		IF GVL_MOTION.STOP_INT THEN
			GVL_MOTION.STATUS.Stop_Int							:= TRUE;
			GVL_MOTION.xCon.Execute_MABS 						:= FALSE;
			GVL_MOTION.yCon.Execute_MABS 						:= FALSE;
			GVL_MOTION.zCon.Execute_MABS 						:= FALSE;
			GVL_MOTION.xCon.Execute_MREL 						:= FALSE;
			GVL_MOTION.yCon.Execute_MREL 						:= FALSE;	
			GVL_MOTION.zCon.Execute_MREL 						:= FALSE;
			GVL_MOTION.xCon.Execute_HALT 						:= TRUE;
			GVL_MOTION.yCon.Execute_HALT 						:= TRUE;
			GVL_MOTION.zCon.Execute_HALT 						:= TRUE;			
				
			GVL_MOTION.InstructionState 						:= 2;
			t5(IN := FALSE);
			
		
		//with no timer pause in between instructions MoveDone stays high long enough to skip an instruction
		//instruction always loaded but queue index is skipped
		ELSIF GVL_MOTION.xOut.MoveDone AND GVL_MOTION.yOut.MoveDone AND GVL_MOTION.zOut.MoveDone THEN //these signals depend on execute MABS/MREL
		
			timer(IN := TRUE, PT := T#1MS);
			
			IF timer.Q THEN
				GVL_MOTION.xCon.Execute_MABS 					:= FALSE;
				GVL_MOTION.xCon.Execute_MREL 					:= FALSE;
				GVL_MOTION.yCon.Execute_MABS 					:= FALSE;
				GVL_MOTION.yCon.Execute_MREL 					:= FALSE;	
				GVL_MOTION.zCon.Execute_MABS 					:= FALSE;
				GVL_MOTION.zCon.Execute_MREL 					:= FALSE;		
				timer(IN := FALSE);
				
				IF GVL_MOTION.CurInstruction < (GVL_MOTION.ScriptEnd - 1) THEN
					GVL_MOTION.CurInstruction 					:= GVL_MOTION.CurInstruction + 1; //queue next instruction
					GVL_MOTION.InstructionState 				:= 0;
					t5(IN := FALSE);
				ELSE
					GVL_MOTION.CurInstruction 					:= 0;
					GVL_MOTION.InstructionState 				:= 0;
					t5(IN := FALSE);
					IF NOT GVL_MOTION.EXT_CTR.CMDLOOP THEN
						IF GVL_MOTION.RUN_INDEX >= GVL_MOTION.EXT_CTR.SCRIPTITERATIONS THEN
							GVL_MOTION.RUN_INDEX				:= 1;
							GVL_MOTION.EXT_CTR.CMDRUN 			:= FALSE;	 //command list executed
						ELSE
							GVL_MOTION.RUN_INDEX				:= GVL_MOTION.RUN_INDEX + 1;	
						END_IF
						
					ELSE
						
						GVL_MOTION.RUN_INDEX					:= GVL_MOTION.RUN_INDEX + 1;
					END_IF
					
				END_IF
				
			END_IF	
			
		END_IF
	
	END_IF
	
	2:
	//state 2: pause motion
	//debounce timer
	t4(IN := TRUE, PT := T#30MS);
	
	
	IF t4.Q THEN
		IF GVL_MOTION.STOP_INT THEN
			GVL_MOTION.STATUS.Stop_Int							:= FALSE; //lamp off
			GVL_MOTION.xCon.Execute_HALT 						:= FALSE;
			GVL_MOTION.yCon.Execute_HALT 						:= FALSE;
			GVL_MOTION.zCon.Execute_HALT 						:= FALSE;
			
			IF GVL_MOTION.Script[GVL_MOTION.CurInstruction].MotionCommand = MotionType.Absolute THEN	
				GVL_MOTION.xCon.Execute_MABS 					:= TRUE;
				GVL_MOTION.yCon.Execute_MABS 					:= TRUE;		
				GVL_MOTION.zCon.Execute_MABS 					:= TRUE;
			
				GVL_MOTION.InstructionState 					:= 1;	
				t4(IN := FALSE);
				
			ELSIF GVL_MOTION.Script[GVL_MOTION.CurInstruction].MotionCommand = MotionType.Relative THEN
				GVL_MOTION.xCon.Execute_MREL 					:= TRUE;
				GVL_MOTION.yCon.Execute_MREL 					:= TRUE;
				GVL_MOTION.zCon.Execute_MREL 					:= TRUE;
			
				GVL_MOTION.InstructionState 			  		:= 1;	
				t4(IN := FALSE);
				
			ELSIF GVL_MOTION.Script[GVL_MOTION.CurInstruction].MotionCommand = MotionType.Time_Wait THEN	
				t2(IN := TRUE, PT := hold);
				GVL_MOTION.InstructionState						:= 3;
			ELSE
				error											:= TRUE;
			END_IF
		
		END_IF
	
	END_IF
	
	3:
	//state 3: timed pause. 
	IF GVL_MOTION.STOP_INT THEN
		GVL_MOTION.STATUS.Stop_Int								:= TRUE; //lamp on
		hold													:= GVL_MOTION.Script[GVL_MOTION.CurInstruction].PauseTime - t2.ET;
		t2(IN := FALSE);
		GVL_MOTION.InstructionState								:= 2;
	ELSIF t2.Q THEN
		t2(IN := FALSE);
		IF GVL_MOTION.CurInstruction < (GVL_MOTION.ScriptEnd - 1) THEN
			GVL_MOTION.CurInstruction 							:= GVL_MOTION.CurInstruction + 1; //queue next instruction
			GVL_MOTION.InstructionState 						:= 0;
					
		ELSE
			GVL_MOTION.CurInstruction 							:= 0;
			GVL_MOTION.InstructionState 						:= 0;
			t5(IN := FALSE);
			IF NOT GVL_MOTION.EXT_CTR.CMDLOOP THEN
				IF GVL_MOTION.RUN_INDEX >= GVL_MOTION.EXT_CTR.SCRIPTITERATIONS THEN
					GVL_MOTION.RUN_INDEX						:= 1;
					GVL_MOTION.EXT_CTR.CMDRUN 					:= FALSE;	 //command list executed
				ELSE
					GVL_MOTION.RUN_INDEX						:= GVL_MOTION.RUN_INDEX + 1;	
				END_IF
				
			ELSE
			
				GVL_MOTION.RUN_INDEX							:= GVL_MOTION.RUN_INDEX + 1;
			END_IF
			
		END_IF
	ELSE
		error													:= TRUE;	
	END_IF
		
END_CASE

END_PROGRAM

// ---- POUs/HomeFixRack.TcPOU
PROGRAM HomeFixRack
VAR
END_VAR

CASE GVL_MOTION.HomingState OF
	0:
	GVL_MOTION.zCon.Execute_HOME			:= TRUE;
	GVL_MOTION.HomingState					:= 1;
	
	1:
	IF GVL_MOTION.zHomeStatus.Done THEN
		GVL_MOTION.zCon.Execute_HOME		:= FALSE;
		GVL_MOTION.yCon.Execute_HOME		:= TRUE;
		GVL_MOTION.HomingState				:= 2;
	END_IF
	
	2:
	IF GVL_MOTION.yHomeStatus.Done THEN
		GVL_MOTION.yCon.Execute_HOME		:= FALSE;
		IF NOT GVL_MOTION.xOut.AxisCoupled THEN
			GVL_MOTION.xCon.ExecuteUncouple	:= FALSE;
			GVL_MOTION.xCon.ExecuteCouple	:= TRUE;
		END_IF
		
		GVL_MOTION.HomingState				:= 3;
	END_IF
	
	3:
	IF GVL_MOTION.xOut.AxisCoupled THEN
		GVL_MOTION.xJogBW					:= TRUE;
		GVL_MOTION.HomingState				:= 4;
	END_IF
	
	4:
	IF GVL_MOTION.xCon.LimNeg OR GVL_MOTION.xcCon.LimNeg THEN
		GVL_MOTION.xJogBW					:= FALSE;
		GVL_MOTION.xCon.SetPosition			:= 5;
		GVL_MOTION.xCon.SetVelocity			:= 50;
		
		GVL_MOTION.HomingState				:= 5;
	
	END_IF
	
	5:
	GVL_MOTION.xCon.Execute_MREL			:= TRUE;
	GVL_MOTION.HomingState					:= 6;	
	
	6:
	IF GVL_MOTION.xOut.MoveDone THEN
		GVL_MOTION.xCon.Execute_MREL		:= FALSE;
		GVL_MOTION.xCon.ExecuteCouple		:= FALSE;
		GVL_MOTION.xCon.ExecuteUncouple 	:= TRUE;
		GVL_MOTION.HomingState				:= 7;
	END_IF
	
	7:
	IF NOT GVL_MOTION.xOut.AxisCoupled THEN
		GVL_MOTION.xCon.Execute_HOME		:= TRUE; 
		GVL_MOTION.HomingState				:= 8;
	END_IF
	
	8:
	IF GVL_MOTION.xHomeStatus.Done THEN
		GVL_MOTION.xCon.Execute_HOME		:= FALSE;
		GVL_MOTION.xcCon.Execute_HOME		:= TRUE;
 		GVL_MOTION.HomingState				:= 9;
	END_IF
	
	9:
	IF GVL_MOTION.xcHomeStatus.Done THEN
		GVL_MOTION.xcCon.Execute_HOME		:= FALSE;
		GVL_MOTION.xCon.ExecuteUncouple 	:= FALSE;
		GVL_MOTION.HomingState				:= 10;
	END_IF
	
	10:
	GVL_MOTION.HomingState					:= 0;
	GVL_MOTION.xCon.ExecuteCouple			:= TRUE;
	GVL_MOTION.AxesLocated					:= TRUE;
	GVL_MOTION.EXT_CTR.CMDHOME				:= FALSE;
END_CASE

END_PROGRAM

// ---- POUs/RackCheck.TcPOU
PROGRAM RackCheck
VAR
	state		:INT	:= 0;
	tempX1		:LREAL;
	tempX2		:LREAL;
	compare		:LREAL;
END_VAR

CASE state OF
	0: //direction of motion unknown
		IF GVL_MOTION.NPNX THEN
			tempX1								:= GVL_MOTION.xOut.PositionOut;
			state								:= 1;
		ELSIF GVL_MOTION.NPNXC THEN	
			tempX1								:= GVL_MOTION.xOut.PositionOut;
			state								:= 2;
		END_IF
		
	1:
		IF GVL_MOTION.NPNXC THEN
			tempX2	:= GVL_MOTION.xOut.PositionOut;
			compare	:= tempX1 - tempX2;
			IF compare > 5 THEN //XC ahead, negative motion
				GVL_MOTION.STATUS.Rack_Err		:= TRUE;
				state							:= 3;
			ELSIF compare < -5 THEN //X ahead, positive motion
				GVL_MOTION.STATUS.Rack_Err		:= TRUE;
				state							:= 3;
			ELSE
				state							:= 0;	
			END_IF
		END_IF	
		
	2:
		IF GVL_MOTION.NPNX THEN
			tempX2								:= GVL_MOTION.xOut.PositionOut;
			compare								:= tempX2 - tempX1;
			IF compare > 5 THEN //XC ahead, positive motion
				GVL_MOTION.STATUS.Rack_Err		:= TRUE;
				state							:= 3;
			ELSIF compare < -5 THEN //X ahead, negative motion
				GVL_MOTION.STATUS.Rack_Err		:= TRUE;
				state							:= 3;
			ELSE
				state							:= 0;	
			END_IF
		END_IF
		
	3: //move X relative by compare
		IF GVL_MOTION.EXT_CTR.CMDFIXRACK AND NOT GVL_MOTION.EXT_CTR.CMDRUN THEN
			GVL_MOTION.xCon.SetPosition			:= compare;
			GVL_MOTION.xCon.ExecuteUncouple		:= TRUE;
			IF NOT GVL_MOTION.xOut.AxisCoupled THEN
				GVL_MOTION.EXT_CTR.CMDFIXRACK	:= FALSE;
				GVL_MOTION.xCon.Execute_MREL	:= TRUE;
				state							:= 4;
			END_IF
		END_IF
	
	4:
		IF GVL_MOTION.xOut.MoveDone THEN
			GVL_MOTION.xCon.Execute_MREL	:= FALSE;
			GVL_MOTION.STATUS.Rack_Err		:= FALSE;
			state							:= 0;
		END_IF
END_CASE

END_PROGRAM

// ---- GlobalTextList.TcGTLO
TEXTLIST GlobalTextList
  803 = '%.0f'
  981 = '%.4f'
  59 = '%4d'
  1444 = '%5d'
  184 = '%s'
  530 = '%t'
  653 = '& Continue From Fault'
  797 = '(Lower Limit)'
  639 = '5'
  56 = '50'
  371 = '500'
  280 = '<- NOT IMPLEMENTED'
  2 = 'A'
  231 = 'ABSOLUTE POSITION'
  461 = 'ACCEL/DECEL'
  34 = 'Accel/Decel'
  466 = 'ACCELERATING'
  532 = 'Actual Position'
  447 = 'Actual Speed'
  575 = 'Add Command to Queue'
  1059 = 'Add Instruction to Script'
  263 = 'AddCMDtoQueue'
  847 = 'AddCMDtoQuue'
  55 = 'Administrator'
  1058 = 'Append Data (single CSV)'
  1775 = 'Axes Located'
  640 = 'Axis to Trigger On'
  687 = 'Axis to Trigger On (NO SICK)'
  2271 = 'B'
  1705 = 'Basin Control'
  458 = 'Basin CTR'
  1413 = 'Basin Set'
  100 = 'BROKEN'
  1205 = 'Capture Data Every X MM'
  869 = 'Capture Data Every X MM/S'
  1220 = 'Clear Data'
  273 = 'Clear Loaded Script'
  848 = 'Clear Queue'
  888 = 'CLICK TO CONTINUE'
  1102 = 'CMD'
  58 = 'CMDtoAdd'
  561 = 'Command'
  312 = 'Command type'
  855 = 'Command Type'
  616 = 'Comment'
  899 = 'Continue From Error'
  293 = 'Continue From Fault'
  313 = 'Continuous Mode'
  1032 = 'Continuous Mode (not for DAQ)'
  101 = 'ContinuousMode'
  425 = 'Couple X Axes'
  416 = 'Current Instruction'
  698 = 'Current Script Run'
  628 = 'DECELERATING'
  1223 = 'Default Basin (Full Area)'
  1420 = 'Delete Last Instruction'
  1786 = 'Delete Loaded Script'
  2013 = 'delete script file'
  140 = 'Delete Script File'
  276 = 'Drive Control'
  485 = 'DRIVE ENABLE'
  614 = 'Drive Error Reset'
  991 = 'E STOP'
  695 = 'ENABLE ALL AXES'
  1622 = 'Enter Comment'
  752 = 'Enter name of basin (no spaces or < > : " / \\ | ? *)'
  1184 = 'Enter Name of Run'
  833 = 'Enter Name of Script'
  326 = 'Enter Name of Script (no spaces or < > : " / \\ | ? *'
  1 = 'Enter Name of Script (no spaces or < > : " / \\ | ? *)'
  1503 = 'Enter Title of Script (no spaces or < > : " / \\ | ? *)'
  958 = 'FAULT RESET'
  745 = 'Fault Reset'
  1527 = 'Fix Rack'
  862 = 'GroupBox'
  665 = 'GVL_MOTION.CommandQueueArray[GVL_MOTION.QueueCur].PauseTime'
  959 = 'Halt'
  241 = 'HaltTime(ms)'
  57 = 'HaltTime(T#XSYMS)'
  95 = 'Home'
  317 = 'Home Both X'
  682 = 'Home Coupled X'
  72 = 'Home Established'
  292 = 'Home X'
  342 = 'Home X (both)'
  733 = 'Home X (not working)'
  1179 = 'Home XYZ'
  846 = 'Home Y'
  185 = 'Home Z'
  689 = 'Homing Routine'
  196 = 'IN POSITION'
  448 = 'IN VELOCITY'
  863 = 'Jog Controls'
  831 = 'k'
  21 = 'Keyence'
  998 = 'Label'
  2027 = 'list'
  420 = 'Locate Hard Stops'
  301 = 'Locate Stops'
  720 = 'Locate Stops NOT IMPLEMENTED'
  712 = 'm'
  245 = 'Main '
  130 = 'Main Sensoor'
  772 = 'Main Sensor'
  605 = 'Main Sensor for DAQ'
  281 = 'Massa'
  319 = 'Motion'
  786 = 'motion cmd'
  1691 = 'Motion CMD'
  545 = 'MOVE ABS EN'
  566 = 'MOVE ACTIVE'
  277 = 'MoveAbsEn'
  632 = 'MOVING'
  1349 = 'Next Instruction'
  633 = 'NOT IMPLEMENTED'
  254 = 'Note: carriage offsets added to these values'
  320 = 'Number of Script Runs'
  1704 = 'Pause'
  457 = 'Pause & WaitOK'
  68 = 'Pause & WaitOK &'
  97 = 'Pause & WaitOK & Continue From Fault'
  105 = 'Pause Motion'
  582 = 'pause time'
  1146 = 'PauseTime'
  818 = 'POSITION'
  473 = 'Position'
  452 = 'Position(AbsorRel'
  926 = 'Position(AbsorRel)'
  996 = 'Position(AbsorRel)(mm)'
  776 = 'PWR Fail'
  787 = 'Rack Error'
  1800 = 'Rackk Error'
  438 = 'Read Script (data/basin/script)'
  634 = 'Read Script (from title)'
  1797 = 'Read Script From File(data/basin/script)'
  419 = 'RELAT'
  676 = 'RELATIVE POSITION'
  572 = 'RESET ALL AXES'
  489 = 'Reset CSV Write'
  162 = 'Reset Enable Error'
  677 = 'REV'
  795 = 'Reverse Couple X'
  719 = 'Run \tQueue'
  999 = 'Run /nQueue'
  256 = 'Run Queue'
  201 = 'RUN QUEUE'
  1126 = 'RUN SCRIPT'
  910 = 'Run Script Continuously'
  785 = 's'
  771 = 'Safe Z Established'
  2090 = 'scriptlist'
  706 = 'Send'
  1909 = 'send list of script names'
  773 = 'send script'
  427 = 'Send To'
  533 = 'Sensor'
  187 = 'Sensors to Record'
  558 = 'Set Basin'
  1079 = 'Set Basin Manually'
  160 = 'Set Safe Z'
  1541 = 'Set Safe Z (lower limit)'
  621 = 'SET SAFE Z FIRST!!'
  1734 = 'Set X'
  53 = 'set x acc'
  1107 = 'set x pos'
  527 = 'set x vel'
  88 = 'Set X Zero'
  717 = 'Set Y'
  1043 = 'set y acc'
  1171 = 'set y pos'
  916 = 'set y vel'
  486 = 'Set Y Zero'
  983 = 'Set Z'
  544 = 'set z pos'
  401 = 'set z vel'
  373 = 'Set Zero'
  604 = 'SICK'
  1746 = 'SICK (X axis)'
  718 = 'SICK (x axis)'
  697 = 'Sonar'
  793 = 'SPEED'
  854 = 'STATIONARY'
  412 = 'STD'
  838 = 'STOP MOTION'
  474 = 'Test for sick (ADS)'
  700 = 'Trigger'
  615 = 'Trigger On'
  1091 = 'Use Basin Coordinates'
  560 = 'Velocity'
  15 = 'VELOCITY CONTROL'
  47 = 'Write Data Test'
  1372 = 'Write Script'
  139 = 'Write Script to File'
  366 = 'X'
  492 = 'x acc'
  129 = 'X Actual Position'
  897 = 'X Actual Speed'
  784 = 'X Coupled Actual Position'
  259 = 'X Coupled Actual Speed'
  901 = 'X Coupled Pos'
  839 = 'X Coupled Spd'
  1675 = 'X Dist to HS'
  2097 = 'X Hard Stop'
  1001 = 'X Max'
  475 = 'X Min'
  511 = 'x pos'
  751 = 'X Position(AbsorRel)(mm)'
  383 = 'x vel'
  885 = 'X Velocity'
  1201 = 'XPos'
  431 = 'xPos'
  255 = 'XVel'
  150 = 'xVel'
  828 = 'xyCMDtoAdd'
  506 = 'xyz motion'
  980 = 'xyzCMDtoAdd'
  1234 = 'xyzMotionCommand'
  906 = 'Y'
  176 = 'y acc'
  746 = 'Y Actual Position'
  547 = 'Y Actual Speed'
  1458 = 'Y Dist to HS'
  1000 = 'Y Hard Stop'
  1376 = 'Y Max'
  215 = 'Y Min'
  982 = 'y pos'
  557 = 'Y Position(AbsorRel)(mm)'
  208 = 'y vel'
  573 = 'Y Velocity'
  559 = 'YPos'
  102 = 'yPos'
  116 = 'YVel'
  8 = 'yVel'
  397 = 'Z'
  509 = 'Z Actual Position'
  504 = 'Z Actual Speed'
  343 = 'z beh'
  432 = 'z brake'
  1751 = 'Z Dist to HS'
  1593 = 'Z Hard Stop'
  631 = 'Z Max'
  1036 = 'Z Min'
  135 = 'z pos'
  972 = 'Z Position(Abs)(mm)'
  662 = 'Z Position(AbsorRel)(mm)'
  125 = 'Z Safe Low'
  1671 = 'z Type'
  636 = 'z vel'
  690 = 'Z Velocity'
  967 = 'zBeh'
  484 = 'zBehavior'
  517 = 'zBehavior (only for xy motion)'
  1119 = 'ZPos'
  49 = 'zPos'
  436 = 'zType'
  1003 = 'ZVel'
  872 = 'zVel'
END_TEXTLIST

// ---- VISUs/visMotorControl.TcVIS
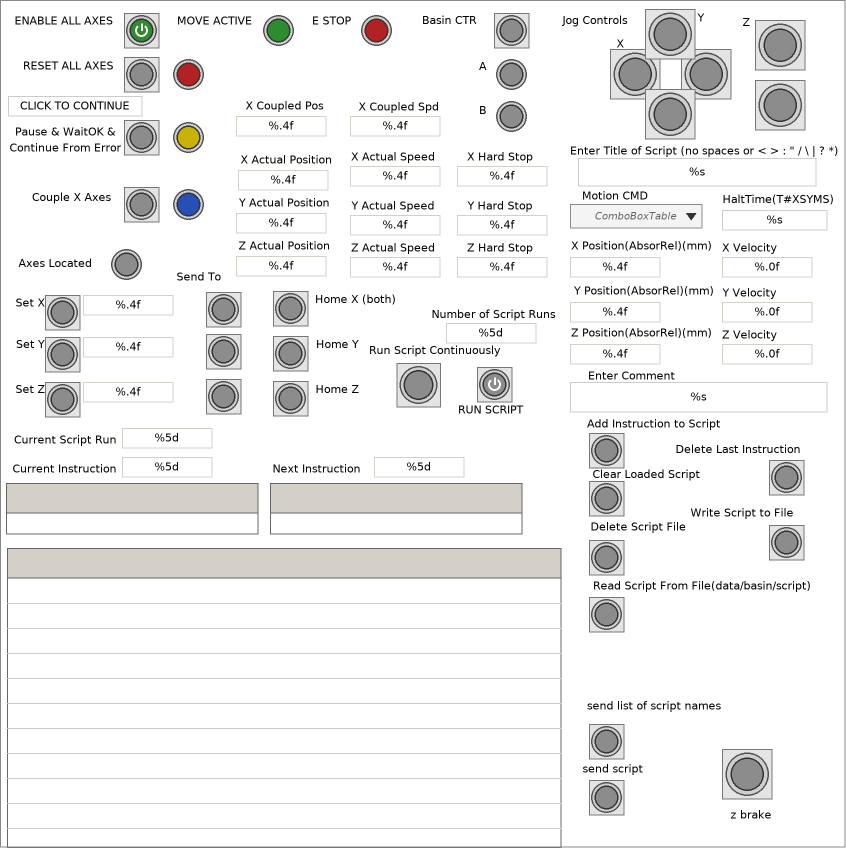
VISUALIZATION visMotorControl  // 846x848
    Label (12,58 113x16), "RESET ALL AXES"
    Label (12,126 107x12), "Pause & WaitOK &"
    Label (9,13 110x16), "ENABLE ALL AXES"
    Textfield (722,257 90x20), "%.0f", text variable: GVL_MOTION.InstructionBuffer.SetXVelocity
        OnMouseClick: write the text variable via InputWithLimits, min 1, max 500, title 'Enter Speed'
    Textfield (570,257 90x20), "%.4f", text variable: GVL_MOTION.InstructionBuffer.SetXPosition
        OnMouseClick: write the text variable via Default, min -200, max 15000
    Label (722,241 55x14), "X Velocity"
    Label (570,238 143x16), "X Position(AbsorRel)(mm)"
    Label (350,149 86x16), "X Actual Speed"
    Label (238,149 97x22), "X Actual Position"
    Textfield (350,166 90x20), "%.4f", text variable: GVL_MOTION.STATUS.xVelOut
    Textfield (238,170 90x20), "%.4f", text variable: GVL_MOTION.STATUS.xPosOut
    ComboBoxTable (570,204 132x24), variable: GVL_MOTION.InstructionBuffer.MotionCommand, data array: GVL_MOTION.xyzCMDSelect
        p1014161805: 4 - 0 + INT#1
        p3854506369: GVL_MOTION.xyzCMDSelect[INDEX]
    Label (564,185 102x22), "Motion CMD"
    PushSwitch (589,433 35x35), variable: GVL_MOTION.EXT_CTR.CMDADD, behaviour: TAP, style: Switch-PushSwitch-Gray
    Label (588,416 132x16), "Add Instruction to Script"
    PushSwitch (589,481 35x35), variable: GVL_MOTION.EXT_CTR.CMDCLR, behaviour: TOGGLE, style: Switch-PushSwitch-Gray
    Label (588,465 117x19), "Clear Loaded Script"
    Label (445,402 91x16), "RUN SCRIPT"
    PowerSwitch (477,367 35x35), variable: GVL_MOTION.EXT_CTR.CMDRUN, behaviour: TOGGLE, style: Switch-PowerSwitch-Gray
    Label (722,192 113x15), "HaltTime(T#XSYMS)"
    Textfield (722,210 105x20), "%s", text variable: GVL_MOTION.InstructionBuffer.pausetime
        OnMouseClick: write the text variable via Default, min 0, max 2000
    Label (554,12 82x17), "Jog Controls"
    PushSwitch (610,49 50x50), variable: GVL_MOTION.xJogBW, behaviour: TAP, style: Switch-PushSwitch-Gray
    PushSwitch (681,49 50x50), variable: GVL_MOTION.xJogFW, behaviour: TAP, style: Switch-PushSwitch-Gray
    Textfield (8,96 134x20), "CLICK TO CONTINUE", invisible if: GVL_MOTION.TxtBxWaitOK
    Lamp1 (171,57 35x35), variable: GVL_MOTION.STATUS.PowerError, style: Lamp-Lamp1-Red
    PushSwitch (45,295 35x35), variable: GVL_MOTION.EXT_CTR.SETXPOS, behaviour: TAP, style: Switch-PushSwitch-Gray
    PushSwitch (273,291 35x35), variable: GVL_MOTION.EXT_CTR.CMDHOMEX, behaviour: TAP, style: Switch-PushSwitch-Gray
    Label (14,295 33x16), "Set X"
    Label (313,291 85x17), "Home X (both)"
    Textfield (570,302 90x20), "%.4f", text variable: GVL_MOTION.InstructionBuffer.SetYPosition
        OnMouseClick: write the text variable via Default, min -200, max 15000
    Label (570,283 148x16), "Y Position(AbsorRel)(mm)"
    Textfield (722,302 90x20), "%.0f", text variable: GVL_MOTION.InstructionBuffer.SetYVelocity
        OnMouseClick: write the text variable via InputWithLimits, min 1, max 500, title 'Enter Speed'
    Label (722,286 55x14), "Y Velocity"
    Label (350,198 86x16), "Y Actual Speed"
    Label (236,192 97x22), "Y Actual Position"
    Textfield (350,215 90x20), "%.4f", text variable: GVL_MOTION.STATUS.yVelOut
    Textfield (236,213 90x20), "%.4f", text variable: GVL_MOTION.STATUS.yPosOut
    PushSwitch (45,337 35x35), variable: GVL_MOTION.EXT_CTR.SETYPOS, behaviour: TAP, style: Switch-PushSwitch-Gray
    Label (14,337 33x15), "Set Y"
    PushSwitch (645,9 50x50), variable: GVL_MOTION.yJogFW, behaviour: TAP, style: Switch-PushSwitch-Gray
    PushSwitch (645,89 50x50), variable: GVL_MOTION.yJogBW, behaviour: TAP, style: Switch-PushSwitch-Gray
    Label (6,141 119x14), "Continue From Error"
    Lamp1 (359,13 35x35), variable: GVL_MOTION.STATUS.eStop, style: Lamp-Lamp1-Red
    Label (300,13 63x16), "E STOP"
    PushSwitch (124,187 35x35), variable: GVL_MOTION.EXT_CTR.CMDCOUPLE, behaviour: TAP, style: Switch-PushSwitch-Gray
    Label (29,192 85x11), "Couple X Axes"
    Lamp1 (171,187 35x35), variable: GVL_MOTION.STATUS.xCoupled, style: Lamp-Lamp1-Blue
    Label (350,99 98x16), "X Coupled Spd"
    Label (236,95 97x22), "X Coupled Pos"
    Textfield (350,116 90x20), "%.4f", text variable: GVL_MOTION.xCOut.VelocityOut
    Textfield (236,116 90x20), "%.4f", text variable: GVL_MOTION.xCOut.PositionOut
    Label (693,9 16x18), "Y"
    Label (603,29 35x30), "X"
    PushSwitch (755,80 50x50), variable: GVL_MOTION.zJogBW, behaviour: TAP, style: Switch-PushSwitch-Gray
    PushSwitch (755,20 50x50), variable: GVL_MOTION.zJogFW, behaviour: TAP, style: Switch-PushSwitch-Gray
    Label (737,13 19x19), "Z"
    Label (350,240 86x16), "Z Actual Speed"
    Label (236,235 97x22), "Z Actual Position"
    Textfield (350,257 90x20), "%.4f", text variable: GVL_MOTION.STATUS.zVelOut
    Textfield (236,256 90x20), "%.4f", text variable: GVL_MOTION.STATUS.zPosOut
    Textfield (446,323 90x20), "%5d", text variable: GVL_MOTION.EXT_CTR.SCRIPTITERATIONS
        OnMouseClick: write the text variable via Default, min 1, title 'Enter Speed'
    Label (428,307 131x15), "Number of Script Runs"
    Label (12,255 87x17), "Axes Located"
    Table (6,483 252x51), data array: GVL_MOTION.Script[GVL_MOTION.CurInstruction]
        p3854506369: GVL_MOTION.Script[GVL_MOTION.CurInstruction].MotionCommand
        p1892666644: GVL_MOTION.Script[GVL_MOTION.CurInstruction].SetXPosition
        p338671338: GVL_MOTION.Script[GVL_MOTION.CurInstruction].SetXVelocity
        p2170511999: GVL_MOTION.Script[GVL_MOTION.CurInstruction].SetXAccel
        p3723444502: GVL_MOTION.Script[GVL_MOTION.CurInstruction].SetYPosition
        p1218418051: GVL_MOTION.Script[GVL_MOTION.CurInstruction].SetYVelocity
        p746581629: GVL_MOTION.Script[GVL_MOTION.CurInstruction].SetYAccel
        p3104783080: GVL_MOTION.Script[GVL_MOTION.CurInstruction].SetZPosition
        p2501879983: GVL_MOTION.Script[GVL_MOTION.CurInstruction].SetZVelocity
        p7306298: GVL_MOTION.Script[GVL_MOTION.CurInstruction].PauseTime
        p1933151965: GVL_MOTION.Script[GVL_MOTION.CurInstruction].Comment
        p511219082: xPos
        p1755163831: xVel
        p2237128397: yPos
        p505689113: yVel
        p4088588272: zPos
        p2243050616: zVel
    Label (368,343 134x15), "Run Script Continuously"
    PushSwitchLed (396,363 45x44), variable: GVL_MOTION.CMDLOOP_INT, behaviour: TOGGLE, style: Switch-PushSwitchLed-Gray
    Label (12,461 105x16), "Current Instruction"
    Textfield (122,457 90x20), "%5d", text variable: GVL_MOTION.CurInstruction
        OnMouseClick: write the text variable via Default
    Table (270,483 252x51), data array: GVL_MOTION.Script[GVL_MOTION.NextInstruction]
        p3854506369: GVL_MOTION.Script[GVL_MOTION.NextInstruction].MotionCommand
        p1892666644: GVL_MOTION.Script[GVL_MOTION.NextInstruction].SetXPosition
        p338671338: GVL_MOTION.Script[GVL_MOTION.NextInstruction].SetXVelocity
        p2170511999: GVL_MOTION.Script[GVL_MOTION.NextInstruction].SetXAccel
        p3723444502: GVL_MOTION.Script[GVL_MOTION.NextInstruction].SetYPosition
        p1218418051: GVL_MOTION.Script[GVL_MOTION.NextInstruction].SetYVelocity
        p746581629: GVL_MOTION.Script[GVL_MOTION.NextInstruction].SetYAccel
        p3104783080: GVL_MOTION.Script[GVL_MOTION.NextInstruction].SetZPosition
        p2501879983: GVL_MOTION.Script[GVL_MOTION.NextInstruction].SetZVelocity
        p7306298: GVL_MOTION.Script[GVL_MOTION.NextInstruction].PauseTime
        p1933151965: GVL_MOTION.Script[GVL_MOTION.NextInstruction].Comment
        p511219082: xPos
        p2237128397: yPos
        p4088588272: zPos
    Label (264,461 105x16), "Next Instruction"
    Textfield (374,457 90x20), "%5d", text variable: GVL_MOTION.NextInstruction
        OnMouseClick: write the text variable via Default
    Textfield (578,158 238x28), "%s", text variable: GVL_MOTION.EXT_CTR.SCRIPTNAME
        OnMouseClick: write GVL_MOTION.EXT_CTR.SCRIPTNAME via Edit
    Label (563,145 283x12), "Enter Title of Script (no spaces or < > : " / \ | ? *)"
    Lamp1 (109,247 35x35), variable: GVL_MOTION.STATUS.AxesLocated, style: Lamp-Lamp1-Gray
    Label (169,13 91x16), "MOVE ACTIVE"
    Textfield (570,344 90x20), "%.4f", text variable: GVL_MOTION.InstructionBuffer.SetZPosition
        OnMouseClick: write the text variable via Default, min -200, max 15000
    Label (570,325 143x16), "Z Position(AbsorRel)(mm)"
    Textfield (722,344 90x20), "%.0f", text variable: GVL_MOTION.InstructionBuffer.SetZVelocity
        OnMouseClick: write the text variable via InputWithLimits, min 1, max 500, title 'Enter Speed'
    Label (722,328 55x14), "Z Velocity"
    Lamp1 (261,13 35x35), variable: GVL_MOTION.STATUS.MoveActive, style: Lamp-Lamp1-Green
    PowerSwitch (124,13 35x35), variable: GVL_MOTION.AXESEN_INT, behaviour: TOGGLE, style: Switch-PowerSwitch-Green
    PushSwitch (124,120 35x35), variable: GVL_MOTION.EXT_CTR.STOP, behaviour: TAP, style: Switch-PushSwitch-Gray
    PushSwitch (124,57 35x35), variable: GVL_MOTION.EXT_CTR.AxesReset, behaviour: TAP, style: Switch-PushSwitch-Gray
    Lamp1 (171,120 35x35), variable: GVL_MOTION.STATUS.STOP_INT, style: Lamp-Lamp1-Yellow
    Label (13,432 105x16), "Current Script Run"
    Textfield (122,428 90x20), "%5d", text variable: GVL_MOTION.RUN_INDEX
        OnMouseClick: write the text variable via Default
    Table (7,548 554x300), data array: GVL_MOTION.Script
        p1014161805: 99 - 0 + INT#1
        p3854506369: GVL_MOTION.Script[INDEX].MotionCommand
        p1892666644: GVL_MOTION.Script[INDEX].SetXPosition
        p338671338: GVL_MOTION.Script[INDEX].SetXVelocity
        p2170511999: GVL_MOTION.Script[INDEX].SetXAccel
        p3723444502: GVL_MOTION.Script[INDEX].SetYPosition
        p1218418051: GVL_MOTION.Script[INDEX].SetYVelocity
        p746581629: GVL_MOTION.Script[INDEX].SetYAccel
        p3104783080: GVL_MOTION.Script[INDEX].SetZPosition
        p2501879983: GVL_MOTION.Script[INDEX].SetZVelocity
        p7306298: GVL_MOTION.Script[INDEX].PauseTime
        p1933151965: GVL_MOTION.Script[INDEX].Comment
        p511219082: xPos
        p1755163831: xVel
        p2237128397: yPos
        p505689113: yVel
        p4088588272: zPos
        p2243050616: zVel
    Textfield (570,382 257x30), "%s", text variable: GVL_MOTION.InstructionBuffer.Comment
        OnMouseClick: write the text variable via Edit
    Label (571,370 121x12), "Enter Comment"
    PushSwitch (769,460 35x35), variable: GVL_MOTION.EXT_CTR.CMDDEL, behaviour: TOGGLE, style: Switch-PushSwitch-Gray
    Label (671,440 134x19), "Delete Last Instruction"
    PushSwitch (769,525 35x35), variable: GVL_MOTION.EXT_CTR.CMDSCRIPTWRITE, behaviour: TOGGLE, style: Switch-PushSwitch-Gray
    Label (691,505 102x16), "Write Script to File"
    PushSwitch (589,597 35x35), variable: GVL_MOTION.EXT_CTR.CMDSCRIPTREAD, behaviour: TOGGLE, style: Switch-PushSwitch-Gray
    Label (588,578 228x16), "Read Script From File(data/basin/script)"
    PushSwitch (494,13 35x35), variable: GVL_MOTION.EXT_CTR.BASINCTR, behaviour: TAP, style: Switch-PushSwitch-Gray
    Label (415,13 69x15), "Basin CTR"
    PushSwitch (45,382 35x35), variable: GVL_MOTION.EXT_CTR.SETZPOS, behaviour: TAP, style: Switch-PushSwitch-Gray
    Label (14,382 33x15), "Set Z"
    Textfield (83,295 90x20), "%.4f", text variable: GVL_MOTION.EXT_CTR.POSX
        OnMouseClick: write the text variable via Default, min -200, max 15000
    Textfield (83,337 90x20), "%.4f", text variable: GVL_MOTION.EXT_CTR.POSY
        OnMouseClick: write the text variable via Default, min -200, max 15000
    Textfield (83,382 90x20), "%.4f", text variable: GVL_MOTION.EXT_CTR.POSZ
        OnMouseClick: write the text variable via Default, min -200, max 15000
    PushSwitch (273,336 35x35), variable: GVL_MOTION.EXT_CTR.CMDHOMEY, behaviour: TAP, style: Switch-PushSwitch-Gray
    Label (313,336 49x17), "Home Y"
    PushSwitch (273,381 35x35), variable: GVL_MOTION.EXT_CTR.CMDHOMEZ, behaviour: TAP, style: Switch-PushSwitch-Gray
    Label (313,381 49x17), "Home Z"
    Label (457,149 86x16), "X Hard Stop"
    Textfield (457,166 90x20), "%.4f", text variable: GVL_MOTION.STATUS.HardStopLocations[0]
    Label (457,198 86x16), "Y Hard Stop"
    Textfield (457,215 90x20), "%.4f", text variable: GVL_MOTION.STATUS.HardStopLocations[1]
    Label (457,240 86x16), "Z Hard Stop"
    Textfield (457,257 90x20), "%.4f", text variable: GVL_MOTION.STATUS.HardStopLocations[2]
    Lamp1 (494,57 35x35), variable: GVL_MOTION.BASINLAMPA, style: Lamp-Lamp1-Gray
    Lamp1 (494,99 35x35), variable: GVL_MOTION.BASINLAMPB, style: Lamp-Lamp1-Gray
    Label (469,59 28x15), "A"
    Label (469,103 28x15), "B"
    PushSwitch (589,724 35x35), variable: GVL_MOTION.EXT_CTR.CMDREQLIST, behaviour: TOGGLE, style: Switch-PushSwitch-Gray
    Label (584,698 140x16), "send list of script names"
    PushSwitch (589,780 35x35), variable: GVL_MOTION.EXT_CTR.CMDREQSCRIPT, behaviour: TOGGLE, style: Switch-PushSwitch-Gray
    Label (578,761 70x16), "send script"
    PushSwitch (589,540 35x35), variable: GVL_MOTION.EXT_CTR.CMDSCRIPTDEL, behaviour: TOGGLE, style: Switch-PushSwitch-Gray
    Label (592,519 93x16), "Delete Script File"
    PushSwitch (722,749 50x50), variable: GVL_MOTION.ED2008O.ED2008_Output.MDP5001_200_DO_Channel_7_Output, behaviour: TOGGLE, style: Switch-PushSwitch-Gray
    Label (722,809 58x12), "z brake"
    PushSwitch (206,292 35x35), variable: GVL_MOTION.EXT_CTR.MOVEX, behaviour: TAP, style: Switch-PushSwitch-Gray
    PushSwitch (206,334 35x35), variable: GVL_MOTION.EXT_CTR.MOVEY, behaviour: TAP, style: Switch-PushSwitch-Gray
    PushSwitch (206,379 35x35), variable: GVL_MOTION.EXT_CTR.MOVEZ, behaviour: TAP, style: Switch-PushSwitch-Gray
    Label (174,269 50x16), "Send To"
END_VISUALIZATION
